INTERFACE I_Device

PROPERTY name : STRING
GET
END_GET
SET
END_SET
END_PROPERTY

END_INTERFACE

(* stored: Version 1.1.0.1
   Itf I_Device: Id {558266e3-a46e-45ac-9221-c39d7967d84c}
   Property name: Id {3264fdf2-c49e-44e5-905e-c4cb9e193020}
   Get Get: Id {8036668f-9561-4dac-b53c-6de5e709244a}
   Set Set: Id {fe4e7028-4d75-4ff3-93da-9f1bc88a88d5} *)
